// TIA Portal V16 export
// export: Created 2021-11-12T13:32:24.4323025Z, ExportSetting WithDefaults, DisplayName Totally Integrated Automation Portal, DisplayVersion V16 Update 3, DisplayName TIA Portal Version Control Interface, DisplayVersion V16 Update 2, DisplayName TIA Portal Openness, DisplayVersion V16 Update 3, DisplayName SINAMICS Startdrive Advanced, DisplayVersion V16 Update 5, DisplayName SINAMICS Startdrive G130, G150, S120, S150, SINAMICS MV, S210, DisplayVersion V16 Update 5, DisplayName SINAMICS Startdrive G110M, G120, G120C, G120D, G120P, G115D, DisplayVersion V16 Update 5, DisplayName STEP 7 Professional, DisplayVersion V16 Update 3, DisplayName STEP 7 Safety, DisplayVersion V16, DisplayName WinCC UA Professional, DisplayVersion V16 Update 3
DATA_BLOCK "STATUS_KAS2"   // DB124
{ S7_Optimized_Access := 'TRUE' }
VERSION : 0.1
// stored: AutoNumber true, DBAccessibleFromOPCUA true, IsOnlyStoredInLoadMemory false, IsRetainMemResEnabled false, IsWriteProtectedInAS false, MemoryReserve 100
   VAR
      xxxxx__BinarySensors__xxxxx : Byte;
      xxxxx__BinaryOthers__xxxxx : Byte;
      xxxxx__AnalogSensors__xxxxx : Byte;
      xxxxx__Drives__xxxxx : Byte;
      xxxxx__Others__xxxxx : Byte;
      NoOfPartsOk : Struct   // Number of OK parts
         Main : "UDT_Status_main";
         Specific : "UDT_PartCounter_Status";
         Error : "UDT_Error01";
      END_STRUCT;
      NoOfPartsNotOk : Struct   // Number of NOK parts
         Main : "UDT_Status_main";
         Specific { S7_SetPoint := 'True'} : "UDT_PartCounter_Status";
         Error { S7_SetPoint := 'True'} : "UDT_Error01";
      END_STRUCT;
      xxxxx__Alarms__xxxxx : Byte;
      LifeBit : Struct   // Communication / Chyba komunikace.
         Main : "UDT_Status_main";
         Specific { S7_SetPoint := 'True'} : "UDT_DI_Mon_Status_specific";
         Error { S7_SetPoint := 'True'} : "UDT_Error01";
      END_STRUCT;
      Saw : Struct   // From saw / Chyba z pily.
         Main : "UDT_Status_main";
         Specific { S7_SetPoint := 'True'} : "UDT_DI_Mon_Status_specific";
         Error { S7_SetPoint := 'True'} : "UDT_Error01";
      END_STRUCT;
      ES : Struct   // E-stop saw 2 / E-stop pila 2.
         Main { S7_SetPoint := 'True'} : "UDT_Status_main";
         Specific { S7_SetPoint := 'True'} : "UDT_DI_Mon_Status_specific";
         Error { S7_SetPoint := 'True'} : "UDT_Error01";
      END_STRUCT;
   END_VAR
BEGIN
END_DATA_BLOCK
